Staubli VAL3: sendJointFbk.pgx

public program sendJointFbk()
begin
  // send message length (prefix)
  nRetVal = sioSet(siTcpIpFbk, nLengthB)
  if (nRetVal == -1)
    putln("Client not connected")
    return
  elseIf (nRetVal < 4)
    popUpMsg("Error while sending prefix")
  endIf

  nBytesSent = size(nLengthB)

  // send message header (msg type, comm type, reply code)
  nRetVal = sioSet(siTcpIpFbk, nMsgTypeB)
  if (nRetVal == -1)
    putln("Client disconnected")
    bStream = false
    return
  elseIf (nRetVal < 4)
    popUpMsg("Error while sending msg type")
  endIf

  nBytesSent = nBytesSent + size(nMsgTypeB)

  nRetVal = sioSet(siTcpIpFbk, nCommTypeB)
  if (nRetVal == -1)
    putln("Client disconnected")
    bStream = false
    return
  elseIf (nRetVal < 4)
    popUpMsg("Error while sending comm type")
  endIf

  nBytesSent = nBytesSent + size(nCommTypeB)

  nRetVal = sioSet(siTcpIpFbk, nReplyCodeB)
  if (nRetVal == -1)
    putln("Client disconnected")
    bStream = false
    return
  elseIf (nRetVal < 4)
    popUpMsg("Error while sending reply code")
  endIf

  nBytesSent = nBytesSent + size(nReplyCodeB)

  // send message body (data)
  // send robotId
  nRetVal = sioSet(siTcpIpFbk, nRobotIdB)
  if (nRetVal == -1)
    putln("client disconnected")
    bStream = false
    return
  elseIf (nRetVal < 4)
    popUpMsg("Error while sending robot ID")
  endIf

  nBytesSent = nBytesSent + size(nRobotIdB)

  // send validFields
  nRetVal = sioSet(siTcpIpFbk, nValidFieldsB)
  if (nRetVal == -1)
    putln("client disconnected")
    bStream = false
    return
  elseIf (nRetVal < 4)
    popUpMsg("Error while sending valid fields")
  endIf

  nBytesSent = nBytesSent + size(nValidFieldsB)

  // send Time
  nRetVal = sioSet(siTcpIpFbk, nTimeB)
  if (nRetVal == -1)
    putln("client disconnected")
    bStream = false
    return
  elseIf (nRetVal < 4)
    popUpMsg("Error while sending timestamp")
  endIf

  nBytesSent = nBytesSent + size(nTimeB)

  // send positions[], velocities[] and accelerations[]
  nRetVal = sioSet(siTcpIpFbk, nPosVelAccB)
  if (nRetVal == -1)
    putln("Client disconnected")
    bStream = false
    return
  elseIf (nRetVal < size(nPosVelAccB))
    popUpMsg("Error while sending msg body")
  endIf

  nBytesSent = nBytesSent + size(nPosVelAccB)

  //put("Joint status sent: ")
  //putln(nBytesSent)
  //bStream = false
end
